(*WARNING WORK-IN-PROGRESS*)
{warning 'DO NOT USE!'}
FUNCTION_BLOCK INTERNAL FB_Hash_Map EXTENDS FB_Collection IMPLEMENTS I_Map
VAR
END_VAR
VAR CONSTANT
	fbBucket_List : FB_Array_List(16) := ();
END_VAR

METHOD FB_init : BOOL
VAR_INPUT
	bInitRetains 	: BOOL; // if TRUE, the retain variables are initialized (warm start / cold start)
	bInCopyCode 	: BOOL;  // if TRUE, the instance afterwards gets moved into the copy code (online change)
END_VAR
END_METHOD

// Gets the value associated with the specified key without remocing it from the dictionary
METHOD Get : I_Map
VAR_INPUT
	Key 			: ANY; // Key used to identify stored value
	Return_Value 	: ANY; // Variable to store requested data 
END_VAR
Get := THIS^;
END_METHOD

// Insert an element with the provided key and value to the dictionary
METHOD Insert : I_Map
VAR_INPUT
	Key 	: ANY; // Key used to identify stored value
	Value 	: ANY; // Value to store in dictionary with key
END_VAR
Insert := THIS^;
END_METHOD

METHOD PROTECTED Populate_Bucket_List : BOOL
VAR_INPUT
	ipList : I_List;
	nCount : T_Capacity;
END_VAR
VAR
	
END_VAR
END_METHOD

// Removes value with the specified key from the dictionary and return that value
METHOD Remove : I_Map
VAR_INPUT
	Key 			: ANY; // Key used to identify stored value
	Return_Value 	: ANY; // Value to store in dictionary with key
END_VAR
Remove := THIS^;
END_METHOD

// Removes the value with the specified key from the dictionary and returns nothing
METHOD Remove_Void : I_Map
VAR_INPUT
	Key 	: ANY; // Key used to identify stored value
END_VAR
Remove_Void := THIS^;
END_METHOD

// Updates the value an element with the provided key and value in the dictionary
METHOD Update : I_Map
VAR_INPUT
	Key 	: ANY; // Key used to identify stored value
	Value 	: ANY; // Value to store in dictionary with key
END_VAR
Update := THIS^;
END_METHOD

END_FUNCTION_BLOCK

(* stored: Version 1.1.0.1, ProductVersion 3.1.4024.4
   POU FB_Hash_Map: Id {a1c8122a-0064-4e5f-8288-29a01c1073f4}, SpecialFunc None
   Folder Protected: Id {3ad05770-7717-4b4c-b69b-af5fadbddb33}
   Method FB_init: Id {c7f11323-ddb4-4746-878e-87028c2b9970}
   Method Get: Id {0a90a1cc-3b89-49b7-969d-f758f548bac2}
   Method Insert: Id {31a4f2f8-93f1-4335-b798-a871e3f75b17}
   Method Populate_Bucket_List: Id {a807a92c-85da-4cef-bd90-412928e9bfc0}
   Method Remove: Id {a60eb9c7-b3ba-473a-be46-bcdac9062fc6}
   Method Remove_Void: Id {faacbc1a-16ad-41ac-a21d-1499c72918fc}
   Method Update: Id {6be44c51-6793-4119-9cdf-ae4e4aeb5234} *)
